FUNCTION_BLOCK FB_manualControl EXTENDS AB_baseController
VAR_INPUT
END_VAR
VAR_OUTPUT
END_VAR
VAR
END_VAR

METHOD control_winch
VAR_INPUT
	stInputs	: ST_inputs_analog;
END_VAR
VAR_OUTPUT
	fMotorValve	: REAL;
END_VAR
fMotorValve := -1.0;
END_METHOD

END_FUNCTION_BLOCK

(* stored: Version 1.1.0.1
   POU FB_manualControl: Id {29d0a2a7-577f-419e-82c9-b14e80532f39}, SpecialFunc None
   Method control_winch: Id {1b80af37-3ec7-473a-b050-6cc7b0491d60} *)
